FUNCTION F_CalculateTransmission : LREAL
VAR_INPUT
    fAbsorptionConstant : LREAL; (* The absorption constant mu, calculated by F_CalculateAbsorptionConstant *)
    fThickness_in_m : LREAL; (* Thickness of the material [m] *)
END_VAR

F_CalculateTransmission := EXP(-fAbsorptionConstant * fThickness_in_m);

END_FUNCTION

(* stored: Version 1.1.0.1, ProductVersion 3.1.4022.18
   POU F_CalculateTransmission: Id {6b6639e0-e794-457e-9110-6d968aadbd26}, SpecialFunc None *)
